FUNCTION_BLOCK FB_StrategyController_noChiller
VAR_INPUT
	ambientState : ST_AmbientState;
	
	//actual temperatures in thermal networks
	cnState : ST_ThermalNetworkState;
	hnltState : ST_ThermalNetworkState;
	hnhtState : ST_ThermalNetworkState;
END_VAR
VAR_OUTPUT	
	cnControl : ST_CoolingNetworkControl;
	hnltControl : ST_HeatingNetworkLowTemperatureControl;	
	hnhtControl : ST_HeatingNetworkHighTemperatureControl;
	hnltCnLinkageControl : ST_HnltCnLinkageControl;
	hnhtHnltLinkageControl : ST_HnhtHnltLinkageControl;
	hnhtCnLinkageControl : ST_HnhtCnLinkageControl;
END_VAR
VAR
	{attribute 'OPC.UA.DA' := '1'}
	localSetParameters : ST_StrategySetParameters;	
	{attribute 'OPC.UA.DA' := '1'}
	localState : ST_StrategyState;	

	//default parameters
	localDefaultParameters : ST_StrategyDefaultParameters;

	//internal variables
	fTargetTemperature_HNHT_Heating : REAL;
	fTargetTemperature_HNHT_Cooling : REAL;
	fTargetTemperature_HNLT_Cooling : REAL;
	fTargetTemperature_HNLT_Heating : REAL;
	fTargetTemperature_CN : REAL;
	aTemperatureLimits_HNHT : ARRAY[1..2] OF REAL;
	aTemperatureLimits_HNLT : ARRAY[1..2] OF REAL;
	aTemperatureLimits_CN : ARRAY[1..2] OF REAL;
	stHNHTCheckDefaultParameters : ST_RangeCheckDefaultParameters := (tTaskCycleTime := GlobalVariables.tCtrlCycleTime_MAIN, tCtrlCycleTime := GlobalVariables.tCtrlCycleTime_MAIN, fRestoreDifference := 5);
	HNHT_Check : FB_RangeCheck := (ST_DefaultParameters := stHNHTCheckDefaultParameters);
	stHNLTCheckDefaultParameters : ST_RangeCheckDefaultParameters := (tTaskCycleTime := GlobalVariables.tCtrlCycleTime_MAIN, tCtrlCycleTime := GlobalVariables.tCtrlCycleTime_MAIN, fRestoreDifference := 5);
	HNLT_Check : FB_RangeCheck := (ST_DefaultParameters := stHNLTCheckDefaultParameters);
	stCNCheckDefaultParameters : ST_RangeCheckDefaultParameters := (tTaskCycleTime := GlobalVariables.tCtrlCycleTime_MAIN, tCtrlCycleTime := GlobalVariables.tCtrlCycleTime_MAIN, fRestoreDifference := 2);
	CN_Check : FB_RangeCheck := (ST_DefaultParameters := stCNCheckDefaultParameters);
	
	
	//controller and variables for high temperature heating network
	fOffset_TargetTemperature_CHP1 : REAL; //not fixed, switches depending on ambient temperature -> see method: ControlHNHT
	fOffset_TargetTemperature_CHP2 : REAL; //not fixed, switches depending on ambient temperature -> see method: ControlHNHT
	Controller_CHP_Prioritization : FB_CTRL_2POINT;
	Controller_CHP_Prioritization_Parameters : ST_CTRL_2POINT_PARAMS;	
	Controller_CHP1_UpperTemperature : FB_CTRL_2POINT; //check upper temperature for turning on chp
	Controller_CHP1_LowerTemperature : FB_CTRL_2POINT; //check lower temperature for turning off chp
	Controller_CHP1_Parameters : ST_CTRL_2POINT_PARAMS;	
	Trigger_CHP1_UpperTemperature : F_TRIG;
	Trigger_CHP1_LowerTemperature : F_TRIG;
	bTrigger_CHP1 : BOOL;
	Controller_CHP2_UpperTemperature : FB_CTRL_2POINT;
	Controller_CHP2_LowerTemperature : FB_CTRL_2POINT;
	Controller_CHP2_Parameters : ST_CTRL_2POINT_PARAMS;
	Trigger_CHP2_UpperTemperature : F_TRIG;
	Trigger_CHP2_LowerTemperature : F_TRIG;
	bTrigger_CHP2 : BOOL;
	Controller_CondensingBoiler : FB_CTRL_2POINT;
	Controller_CondensingBoiler_Parameters : ST_CTRL_2POINT_PARAMS;
	Controller_VSI_Loading_Permission : FB_CTRL_2POINT;
	Controller_VSI_Loading_Permission_Parameters : ST_CTRL_2POINT_PARAMS;
	Controller_VSI_Unloading_Permission : FB_CTRL_2POINT;
	Controller_VSI_Unloading_Permission_Parameters : ST_CTRL_2POINT_PARAMS;
	Controller_Buffer_VSI_Unloading : FB_CTRL_2POINT;
	Controller_Buffer_VSI_Unloading_Parameters : ST_CTRL_2POINT_PARAMS;
	Controller_StaticHeating : FB_CTRL_2POINT;
	Controller_StaticHeating_Parameters : ST_CTRL_2POINT_PARAMS;
	
	//controllers and variables for low temperature heating network
	Controller_OuterCapillaryTubeMats : FB_CTRL_2POINT;
	Controller_OuterCapillaryTubeMats_Parameters : ST_CTRL_2POINT_PARAMS;
	Controller_OuterCapillaryTubeMats_Permission : FB_CTRL_2POINT;
	Controller_OuterCapillaryTubeMats_Permission_Parameters : ST_CTRL_2POINT_PARAMS;
	fOffset_TargetTemperature_OuterCapillaryTubeMats_Cooling : REAL := 1;	
	fOffset_OuterCapillaryTubeMats_Permission : REAL := 10;
	
	Controller_HVFA_HNLT_HVFALoadingPermission : FB_CTRL_2POINT;
	Controller_HVFA_HNLT_HVFALoadingPermission_Parameters : ST_CTRL_2POINT_PARAMS;
	Controller_HVFA_HNLT_HVFAUnloadingPermission : FB_CTRL_2POINT;
	Controller_HVFA_HNLT_HVFAUnloadingPermission_Parameters : ST_CTRL_2POINT_PARAMS;
	Controller_Buffer_HVFA_HNLT_HVFAUnloading : FB_CTRL_2POINT;
	Controller_Buffer_HVFA_HNLT_HVFAUnloading_Parameters : ST_CTRL_2POINT_PARAMS;
	Controller_Buffer_HVFA_HNLT_HVFALoading : FB_CTRL_2POINT;
	Controller_Buffer_HVFA_HNLT_HVFALoading_Parameters : ST_CTRL_2POINT_PARAMS;
	Controller_HVFA_HNLT_Recooling : FB_CTRL_2POINT;
	Controller_HVFA_HNLT_Recooling_Parameters : ST_CTRL_2POINT_PARAMS;
	fOffset_TargetTemperature_HVFA_HNLT_Heating : REAL := 1;
	fOffset_HVFA_HNLT_Recooling : REAL := 2;
		
	
	//controllers and variables for cooling network
	fOffset_TargetTemperature_eChiller : REAL := 0.5;	
	fOffset_TargetTemperature_HVFA_CN : REAL := 1;
	fOffset_TargetTemperature_HVFA_CN_Permission : REAL := 2.5;
	Controller_eChiller : FB_CTRL_2POINT;
	Controller_eChiller_Parameters : ST_CTRL_2POINT_PARAMS;	
	Controller_HVFA_CN_LoadingPermission : FB_CTRL_2POINT;
	Controller_HVFA_CN_LoadingPermission_Parameters : ST_CTRL_2POINT_PARAMS;
	Controller_HVFA_CN_UnloadingPermission : FB_CTRL_2POINT;
	Controller_HVFA_CN_UnloadingPermission_Parameters : ST_CTRL_2POINT_PARAMS;
	Controller_Buffer_HVFA_CN_Unloading : FB_CTRL_2POINT;
	Controller_Buffer_HVFA_CN_Unloading_Parameters : ST_CTRL_2POINT_PARAMS;

	//controllers and variables for hnht and hnlt linkage
	Controller_HeatExchanger1 : FB_CTRL_2POINT;
	Controller_HeatExchanger1_Parameters : ST_CTRL_2POINT_PARAMS;
	fOffset_TargetTemperature_HeatExchanger1 : REAL := 2;
	Controller_HeatPump_HNHT : FB_CTRL_2POINT;
	Controller_HeatPump_HNHT_Parameters : ST_CTRL_2POINT_PARAMS;
	fOffset_TargetTemperature_HeatPump_HNHT : REAL := 1;
	Controller_HeatPump_HNHT_Permission : FB_CTRL_2POINT;
	Controller_HeatPump_HNHT_Permission_Parameters : ST_CTRL_2POINT_PARAMS;
	fOffset_TargetTemperature_HeatPump_HNHT_Permission : REAL := 1;
	
	//controllers and variables for hnlt and cn linkage
	fOffset_TargetTemperature_HeatPump : REAL;
	Controller_HeatPump : FB_CTRL_2POINT;
	Controller_HeatPump_Parameters : ST_CTRL_2POINT_PARAMS;		

	//clock
	stDefaultParameters_Clock : ST_ClockDefaultParameters := (tTaskCycleTime := GlobalVariables.tCtrlCycleTime_MAIN, tCtrlCycleTime := T#1M);
	Clock : FB_Clock := (ST_DefaultParameters := stDefaultParameters_Clock);
END_VAR

Clock();
AmbientControl();
SetTemperatures();
ControlCN();
ControlHNLT();
ControlHNHT();
ControlHnltCnLinkage();
ControlHnhtHnltLinkage();
SetState();

METHOD AmbientControl : BOOL
VAR_INPUT
END_VAR
//check for heating or cooling mode
IF Clock.stClockState.sintMonth>4 AND Clock.stClockState.sintMonth<10 THEN
	//heating mode
	hnltCnLinkageControl.bHeatingMode := FALSE;
	hnhtCnLinkageControl.bHeatingMode := FALSE;
ELSE
	//cooling mode	
	hnltCnLinkageControl.bHeatingMode := TRUE;
	hnhtCnLinkageControl.bHeatingMode := TRUE;
END_IF
END_METHOD

METHOD ControlCN : BOOL
VAR_INPUT
END_VAR
//set hysteresis parameters for two-point controllers in cooling network
Controller_eChiller_Parameters.fHysteresisRange := 7;
Controller_eChiller_Parameters.tCtrlCycleTime := GlobalVariables.tCtrlCycleTime_MAIN;
Controller_eChiller_Parameters.tTaskCycleTime := GlobalVariables.tTaskCycleTime_MAIN;

//permission to load storage depending on upper hvfa storage temperature
Controller_HVFA_CN_LoadingPermission_Parameters.fHysteresisRange := 1;
Controller_HVFA_CN_LoadingPermission_Parameters.tCtrlCycleTime := GlobalVariables.tCtrlCycleTime_MAIN;
Controller_HVFA_CN_LoadingPermission_Parameters.tTaskCycleTime := GlobalVariables.tTaskCycleTime_MAIN;

//permission to unload storage depending on upper hvfa storage temperature
Controller_HVFA_CN_UnloadingPermission_Parameters.fHysteresisRange := 1;
Controller_HVFA_CN_UnloadingPermission_Parameters.tCtrlCycleTime := GlobalVariables.tCtrlCycleTime_MAIN;
Controller_HVFA_CN_UnloadingPermission_Parameters.tTaskCycleTime := GlobalVariables.tTaskCycleTime_MAIN;

//hysteresis for unloading hvfa storage depending on buffer storage temperature
Controller_Buffer_HVFA_CN_Unloading_Parameters.fHysteresisRange := 2;
Controller_Buffer_HVFA_CN_Unloading_Parameters.tCtrlCycleTime := GlobalVariables.tCtrlCycleTime_MAIN;
Controller_Buffer_HVFA_CN_Unloading_Parameters.tTaskCycleTime := GlobalVariables.tTaskCycleTime_MAIN;

//control eChiller
Controller_eChiller(fSetpointValue := cnState.fMidTemperature,
	fActualValue := fTargetTemperature_CN-fOffset_TargetTemperature_eChiller,
	eMode := eCTRL_MODE_ACTIVE,
	stParams := Controller_eChiller_Parameters);

//control hvfa storage loading permission 
Controller_HVFA_CN_LoadingPermission(fSetpointValue := cnState.fUpperTemperature_ActiveStorage,
	fActualValue := fTargetTemperature_CN-fOffset_TargetTemperature_HVFA_CN_Permission,
	eMode := eCTRL_MODE_ACTIVE,
	stParams := Controller_HVFA_CN_LoadingPermission_Parameters);
	
//control hvfa storage unloading permission 
Controller_HVFA_CN_UnloadingPermission(fSetpointValue := fTargetTemperature_CN-fOffset_TargetTemperature_HVFA_CN_Permission,
	fActualValue := cnState.fLowerTemperature_ActiveStorage,
	eMode := eCTRL_MODE_ACTIVE,
	stParams := Controller_HVFA_CN_UnloadingPermission_Parameters);
	
//unloading permission buffer HVFA
Controller_Buffer_HVFA_CN_Unloading(fSetpointValue := cnState.fMidTemperature,
	fActualValue := fTargetTemperature_CN+fOffset_TargetTemperature_HVFA_CN,
	eMode := eCTRL_MODE_ACTIVE,
	stParams := Controller_Buffer_HVFA_CN_Unloading_Parameters);
	
IF Clock.stClockState.sintMonth>4 AND Clock.stClockState.sintMonth<10 THEN
	cnControl.bSetStatusOn_eChiller := TRUE;
	cnControl.bSetStatusOn_HVFASystem := FALSE;
	cnControl.bLoading_HVFASystem := FALSE;
ELSE
	cnControl.bSetStatusOn_eChiller := Controller_eChiller.bOut;
	cnControl.bSetStatusOn_HVFASystem := (Controller_Buffer_HVFA_CN_Unloading.bOut AND Controller_HVFA_CN_UnloadingPermission.bOut) OR ((cnControl.bSetStatusOn_eChiller) AND NOT Controller_Buffer_HVFA_CN_Unloading.bOut AND Controller_HVFA_CN_LoadingPermission.bOut); 
	cnControl.bLoading_HVFASystem := NOT (Controller_Buffer_HVFA_CN_Unloading.bOut AND Controller_HVFA_CN_UnloadingPermission.bOut);
END_IF

cnControl.bSetStatusOn_eChiller := FALSE; //strategy without eChiller
cnControl.bSetStatusOn_HVFASystem := FALSE;
cnControl.bLoading_HVFASystem := FALSE;


//cnControl.bSetStatusOn_HVFASystem := FALSE;
//cnControl.bLoading_HVFASystem := FALSE;
END_METHOD

METHOD ControlHNHT : BOOL
VAR_INPUT
END_VAR
VAR
END_VAR
//set hysteresis parameters for two-point controllers in high temperature heating network
Controller_CHP_Prioritization_Parameters.fHysteresisRange := 4;
Controller_CHP_Prioritization_Parameters.tCtrlCycleTime := GlobalVariables.tCtrlCycleTime_MAIN;
Controller_CHP_Prioritization_Parameters.tTaskCycleTime := GlobalVariables.tTaskCycleTime_MAIN;

Controller_CHP1_Parameters.tCtrlCycleTime := GlobalVariables.tCtrlCycleTime_MAIN;
Controller_CHP1_Parameters.tTaskCycleTime := GlobalVariables.tTaskCycleTime_MAIN;
Controller_CHP2_Parameters.tCtrlCycleTime := GlobalVariables.tCtrlCycleTime_MAIN;
Controller_CHP2_Parameters.tTaskCycleTime := GlobalVariables.tTaskCycleTime_MAIN;

Controller_CondensingBoiler_Parameters.fHysteresisRange := 12;
Controller_CondensingBoiler_Parameters.tCtrlCycleTime := GlobalVariables.tCtrlCycleTime_MAIN;
Controller_CondensingBoiler_Parameters.tTaskCycleTime := GlobalVariables.tTaskCycleTime_MAIN;

Controller_Buffer_VSI_Unloading_Parameters.fHysteresisRange := 4;
Controller_Buffer_VSI_Unloading_Parameters.tCtrlCycleTime := GlobalVariables.tCtrlCycleTime_MAIN;
Controller_Buffer_VSI_Unloading_Parameters.tTaskCycleTime := GlobalVariables.tTaskCycleTime_MAIN;

Controller_VSI_Unloading_Permission_Parameters.fHysteresisRange := 4;
Controller_VSI_Unloading_Permission_Parameters.tCtrlCycleTime := GlobalVariables.tCtrlCycleTime_MAIN;
Controller_VSI_Unloading_Permission_Parameters.tTaskCycleTime := GlobalVariables.tTaskCycleTime_MAIN;

Controller_VSI_Loading_Permission_Parameters.fHysteresisRange := 4;
Controller_VSI_Loading_Permission_Parameters.tCtrlCycleTime := GlobalVariables.tCtrlCycleTime_MAIN;
Controller_VSI_Loading_Permission_Parameters.tTaskCycleTime := GlobalVariables.tTaskCycleTime_MAIN;

Controller_StaticHeating_Parameters.fHysteresisRange := 4;
Controller_StaticHeating_Parameters.tCtrlCycleTime := GlobalVariables.tCtrlCycleTime_MAIN;
Controller_StaticHeating_Parameters.tTaskCycleTime := GlobalVariables.tTaskCycleTime_MAIN;

Controller_CHP_Prioritization(fSetpointValue := 15,
	fActualValue := ambientState.fOutsideTemperature_Mean,
	eMode := eCTRL_MODE_ACTIVE,
	stParams := Controller_CHP_Prioritization_Parameters);
IF Controller_CHP_Prioritization.bOut THEN
	//prioritize large CHP (CHP2) during cold temperatures
	Controller_CHP1_Parameters.fHysteresisRange := 14;
	Controller_CHP2_Parameters.fHysteresisRange := 12;
	fOffset_TargetTemperature_CHP1 := 1;
	fOffset_TargetTemperature_CHP2 := 0;
ELSE
	//prioritize large CHP (CHP2) during cold temperatures
	Controller_CHP1_Parameters.fHysteresisRange := 12;
	Controller_CHP2_Parameters.fHysteresisRange := 14;	
	fOffset_TargetTemperature_CHP1 := 0;
	fOffset_TargetTemperature_CHP2 := 1;	
END_IF

//start when upper temperature too cold and stop when lower temperature too hot
Controller_CHP1_UpperTemperature(fSetpointValue := fTargetTemperature_HNHT_Heating-fOffset_TargetTemperature_CHP1,
	fActualValue := hnhtState.fUpperTemperature,
	eMode := eCTRL_MODE_ACTIVE,
	stParams := Controller_CHP1_Parameters);
Controller_CHP1_LowerTemperature(fSetpointValue := fTargetTemperature_HNHT_Heating-fOffset_TargetTemperature_CHP1,
	fActualValue := hnhtState.fLowerTemperature,
	eMode := eCTRL_MODE_ACTIVE,
	stParams := Controller_CHP1_Parameters);
Trigger_CHP1_UpperTemperature(CLK := Controller_CHP1_UpperTemperature.bOut);
Trigger_CHP1_LowerTemperature(CLK := Controller_CHP1_LowerTemperature.bOut);
IF Trigger_CHP1_UpperTemperature.Q THEN
	bTrigger_CHP1 := TRUE;
END_IF
IF Trigger_CHP1_LowerTemperature.Q THEN
	bTrigger_CHP1 := FALSE;
END_IF
hnhtControl.bSetStatusOn_CHP1 := Controller_CHP1_UpperTemperature.bOut OR (Controller_CHP1_LowerTemperature.bOut AND bTrigger_CHP1);

//start when upper temperature too cold and stop when lower temperature too hot
Controller_CHP2_UpperTemperature(fSetpointValue := fTargetTemperature_HNHT_Heating-fOffset_TargetTemperature_CHP2,
	fActualValue := hnhtState.fUpperTemperature,
	eMode := eCTRL_MODE_ACTIVE,
	stParams := Controller_CHP2_Parameters);
Controller_CHP2_LowerTemperature(fSetpointValue := fTargetTemperature_HNHT_Heating-fOffset_TargetTemperature_CHP2,
	fActualValue := hnhtState.fLowerTemperature,
	eMode := eCTRL_MODE_ACTIVE,
	stParams := Controller_CHP2_Parameters);
Trigger_CHP2_UpperTemperature(CLK := Controller_CHP2_UpperTemperature.bOut);
Trigger_CHP2_LowerTemperature(CLK := Controller_CHP2_LowerTemperature.bOut);
IF Trigger_CHP2_UpperTemperature.Q THEN
	bTrigger_CHP2 := TRUE;
END_IF
IF Trigger_CHP2_LowerTemperature.Q THEN
	bTrigger_CHP2 := FALSE;
END_IF
hnhtControl.bSetStatusOn_CHP2 := Controller_CHP2_UpperTemperature.bOut OR (Controller_CHP2_LowerTemperature.bOut AND bTrigger_CHP2);

Controller_CondensingBoiler(fSetpointValue := fTargetTemperature_HNHT_Heating,
	fActualValue := hnhtState.fUpperTemperature,
	eMode := eCTRL_MODE_ACTIVE,
	stParams := Controller_CondensingBoiler_Parameters);
hnhtControl.bSetStatusOn_CondensingBoiler := Controller_CondensingBoiler.bOut;

//buffer storage asks VSI for unloading when buffer storage temperature falls below limit
Controller_Buffer_VSI_Unloading(fSetpointValue := fTargetTemperature_HNHT_Heating,
	fActualValue := hnhtState.fUpperTemperature,
	eMode := eCTRL_MODE_ACTIVE,
	stParams := Controller_Buffer_VSI_Unloading_Parameters);

//VSI storage may only be unloaded when upper temperature is between limits for unloading
Controller_VSI_Unloading_Permission(fSetpointValue := hnhtState.fUpperTemperature_ActiveStorage,
	fActualValue := fTargetTemperature_HNHT_Heating,
	eMode := eCTRL_MODE_ACTIVE,
	stParams := Controller_VSI_Unloading_Permission_Parameters);
	
//VSI storage may only be loaded when lower temperature is between limits for loading
Controller_VSI_Loading_Permission(fSetpointValue := fTargetTemperature_HNHT_Heating,
	fActualValue := hnhtState.fLowerTemperature_ActiveStorage,
	eMode := eCTRL_MODE_ACTIVE,
	stParams := Controller_VSI_Loading_Permission_Parameters);
	
hnhtControl.bSetStatusOn_VSIStorage := (Controller_Buffer_VSI_Unloading.bOut AND Controller_VSI_Unloading_Permission.bOut) OR ((hnhtControl.bSetStatusOn_CHP1 OR hnhtControl.bSetStatusOn_CHP2) AND NOT Controller_Buffer_VSI_Unloading.bOut AND Controller_VSI_Loading_Permission.bOut); 
hnhtControl.bLoading_VSISystem := NOT (Controller_Buffer_VSI_Unloading.bOut AND Controller_VSI_Unloading_Permission.bOut);

//condensing boiler is switched if network temperature falls below critical temperature limit
Controller_StaticHeating(fSetpointValue := 15,
	fActualValue := ambientState.fOutsideTemperature,
	eMode := eCTRL_MODE_ACTIVE,
	stParams := Controller_StaticHeating_Parameters);
hnhtControl.bSetStatusOn_StaticHeating := Controller_StaticHeating.bOut;
END_METHOD

METHOD ControlHnhtHnltLinkage : BOOL
VAR_INPUT
END_VAR
Controller_HeatExchanger1_Parameters.fHysteresisRange := 8;
Controller_HeatExchanger1_Parameters.tCtrlCycleTime := GlobalVariables.tCtrlCycleTime_MAIN;
Controller_HeatExchanger1_Parameters.tTaskCycleTime := GlobalVariables.tTaskCycleTime_MAIN;

Controller_HeatPump_HNHT_Parameters.fHysteresisRange := 10;
Controller_HeatPump_HNHT_Parameters.tCtrlCycleTime := GlobalVariables.tCtrlCycleTime_MAIN;
Controller_HeatPump_HNHT_Parameters.tTaskCycleTime := GlobalVariables.tTaskCycleTime_MAIN;

Controller_HeatPump_HNHT_Permission_Parameters.fHysteresisRange := 4;
Controller_HeatPump_HNHT_Permission_Parameters.tCtrlCycleTime := GlobalVariables.tCtrlCycleTime_MAIN;
Controller_HeatPump_HNHT_Permission_Parameters.tTaskCycleTime := GlobalVariables.tTaskCycleTime_MAIN;

//control heat exchanger 1
Controller_HeatExchanger1(fSetpointValue := fTargetTemperature_HNLT_Heating-fOffset_TargetTemperature_HeatExchanger1,
	fActualValue := hnltState.fMidTemperature,
	eMode := eCTRL_MODE_ACTIVE,
	stParams := Controller_HeatExchanger1_Parameters);
hnhtHnltLinkageControl.bSetStatusOn_HeatExchanger1 := Controller_HeatExchanger1.bOut;

//control heat pump hnht
Controller_HeatPump_HNHT(fSetpointValue := fTargetTemperature_HNHT_Heating+fOffset_TargetTemperature_HeatPump_HNHT,
	fActualValue := hnhtState.fUpperTemperature,
	eMode := eCTRL_MODE_ACTIVE,
	stParams := Controller_HeatPump_HNHT_Parameters);
	
Controller_HeatPump_HNHT_Permission(fSetpointValue := hnltState.fMidTemperature,
	fActualValue := fTargetTemperature_HNLT_Cooling+fOffset_TargetTemperature_HeatPump_HNHT_Permission,
	eMode := eCTRL_MODE_ACTIVE,
	stParams := Controller_HeatPump_HNHT_Permission_Parameters);	
	
// HP currently only able to reach 65°C flow temperature (hard-coded HP-internal)
// IF localSetParameters.bProductionModeActivated THEN
// 	hnhtHnltLinkageControl.bSetStatusOn_HeatPump := FALSE;
// ELSE
// 	hnhtHnltLinkageControl.bSetStatusOn_HeatPump := Controller_HeatPump_HNHT.bOut AND Controller_HeatPump_HNHT_Permission.bOut;
// END_IF

// When using a heating target temp of 60 °C in production mode the heat pump can be used in both operating modes
hnhtHnltLinkageControl.bSetStatusOn_HeatPump := Controller_HeatPump_HNHT.bOut AND Controller_HeatPump_HNHT_Permission.bOut;
END_METHOD

METHOD ControlHNLT : BOOL
VAR_INPUT
END_VAR
//set hysteresis parameters for two-point controllers in cooling network
Controller_OuterCapillaryTubeMats_Parameters.fHysteresisRange := 6;
Controller_OuterCapillaryTubeMats_Parameters.tCtrlCycleTime := GlobalVariables.tCtrlCycleTime_MAIN;
Controller_OuterCapillaryTubeMats_Parameters.tTaskCycleTime := GlobalVariables.tTaskCycleTime_MAIN;

Controller_OuterCapillaryTubeMats_Permission_Parameters.fHysteresisRange := 6;
Controller_OuterCapillaryTubeMats_Permission_Parameters.tCtrlCycleTime := GlobalVariables.tCtrlCycleTime_MAIN;
Controller_OuterCapillaryTubeMats_Permission_Parameters.tTaskCycleTime := GlobalVariables.tTaskCycleTime_MAIN;


//control strategy for cooling network - fSetpointValue and fActualValue are changed for cooling applications
Controller_OuterCapillaryTubeMats(fSetpointValue := hnltState.fMidTemperature,
	fActualValue := fTargetTemperature_HNLT_Cooling+fOffset_TargetTemperature_OuterCapillaryTubeMats_Cooling,
	eMode := eCTRL_MODE_ACTIVE,
	stParams := Controller_OuterCapillaryTubeMats_Parameters);

//permission controller to ensure that network ist not heated up if ambient temperature is too high
Controller_OuterCapillaryTubeMats_Permission(fSetpointValue := fTargetTemperature_HNLT_Cooling-fOffset_OuterCapillaryTubeMats_Permission,
	fActualValue := ambientState.fOutsideTemperature,
	eMode := eCTRL_MODE_ACTIVE,
	stParams := Controller_OuterCapillaryTubeMats_Permission_Parameters);

//control hvfa storage
//set hysteresis parameters for two-point controllers in low temperature heating network

Controller_Buffer_HVFA_HNLT_HVFAUnloading_Parameters.fHysteresisRange := 6;
Controller_Buffer_HVFA_HNLT_HVFAUnloading_Parameters.tCtrlCycleTime := GlobalVariables.tCtrlCycleTime_MAIN;
Controller_Buffer_HVFA_HNLT_HVFAUnloading_Parameters.tTaskCycleTime := GlobalVariables.tTaskCycleTime_MAIN;

Controller_Buffer_HVFA_HNLT_HVFALoading_Parameters.fHysteresisRange := 4;
Controller_Buffer_HVFA_HNLT_HVFALoading_Parameters.tCtrlCycleTime := GlobalVariables.tCtrlCycleTime_MAIN;
Controller_Buffer_HVFA_HNLT_HVFALoading_Parameters.tTaskCycleTime := GlobalVariables.tTaskCycleTime_MAIN;

Controller_HVFA_HNLT_Recooling_Parameters.fHysteresisRange := 4;
Controller_HVFA_HNLT_Recooling_Parameters.tCtrlCycleTime := GlobalVariables.tCtrlCycleTime_MAIN;
Controller_HVFA_HNLT_Recooling_Parameters.tTaskCycleTime := GlobalVariables.tTaskCycleTime_MAIN;

Controller_HVFA_HNLT_HVFAUnloadingPermission_Parameters.fHysteresisRange := 4;
Controller_HVFA_HNLT_HVFAUnloadingPermission_Parameters.tCtrlCycleTime := GlobalVariables.tCtrlCycleTime_MAIN;
Controller_HVFA_HNLT_HVFAUnloadingPermission_Parameters.tTaskCycleTime := GlobalVariables.tTaskCycleTime_MAIN;

Controller_HVFA_HNLT_HVFALoadingPermission_Parameters.fHysteresisRange := 4;
Controller_HVFA_HNLT_HVFALoadingPermission_Parameters.tCtrlCycleTime := GlobalVariables.tCtrlCycleTime_MAIN;
Controller_HVFA_HNLT_HVFALoadingPermission_Parameters.tTaskCycleTime := GlobalVariables.tTaskCycleTime_MAIN;

//buffer storage asks HVFA_HNLT for unloading when buffer storage temperature falls below limit
Controller_Buffer_HVFA_HNLT_HVFAUnloading(fSetpointValue := fTargetTemperature_HNLT_Heating-fOffset_TargetTemperature_HVFA_HNLT_Heating,
	fActualValue := hnltState.fMidTemperature,
	eMode := eCTRL_MODE_ACTIVE,
	stParams := Controller_Buffer_HVFA_HNLT_HVFAUnloading_Parameters);
	
//buffer storage asks HVFA_HNLT for loading when buffer storage temperature rises above limit
Controller_Buffer_HVFA_HNLT_HVFALoading(fSetpointValue := hnltState.fMidTemperature,
	fActualValue := fTargetTemperature_HNLT_Cooling,
	eMode := eCTRL_MODE_ACTIVE,
	stParams := Controller_Buffer_HVFA_HNLT_HVFALoading_Parameters);

//hvfa storage may only be unloaded when upper temperature is between limits for unloading
Controller_HVFA_HNLT_HVFAUnloadingPermission(fSetpointValue := hnltState.fLowerTemperature_ActiveStorage,
	fActualValue := fTargetTemperature_HNLT_Heating,
	eMode := eCTRL_MODE_ACTIVE,
	stParams := Controller_HVFA_HNLT_HVFAUnloadingPermission_Parameters);
	
//hvfa storage may only be loaded when lower temperature is between limits for loading
Controller_HVFA_HNLT_HVFALoadingPermission(fSetpointValue := fTargetTemperature_HNLT_Cooling,
	fActualValue := hnltState.fLowerTemperature_ActiveStorage,
	eMode := eCTRL_MODE_ACTIVE,
	stParams := Controller_HVFA_HNLT_HVFALoadingPermission_Parameters);

//enable hvfa recooling during low temperature times in summer months	
Controller_HVFA_HNLT_Recooling(fSetpointValue := hnltState.fLowerTemperature_ActiveStorage,
	fActualValue := fTargetTemperature_HNLT_Cooling-fOffset_HVFA_HNLT_Recooling,
	eMode := eCTRL_MODE_ACTIVE,
	stParams := Controller_HVFA_HNLT_Recooling_Parameters);
	
IF hnltCnLinkageControl.bHeatingMode THEN
	hnltControl.bSetStatusOn_HVFASystem := (Controller_HVFA_HNLT_HVFALoadingPermission.bOut AND Controller_Buffer_HVFA_HNLT_HVFALoading.bOut) OR (Controller_HVFA_HNLT_HVFAUnloadingPermission.bOut AND Controller_Buffer_HVFA_HNLT_HVFAUnloading.bOut);
	hnltControl.bLoading_HVFASystem := Controller_HVFA_HNLT_HVFALoadingPermission.bOut AND Controller_Buffer_HVFA_HNLT_HVFALoading.bOut;
	hnltControl.bSetStatusOn_OuterCapillaryTubeMats := Controller_OuterCapillaryTubeMats.bOut AND Controller_OuterCapillaryTubeMats_Permission.bOut;
ELSE
	hnltControl.bSetStatusOn_HVFASystem := ((Controller_HVFA_HNLT_HVFALoadingPermission.bOut AND Controller_Buffer_HVFA_HNLT_HVFALoading.bOut) OR (Controller_HVFA_HNLT_HVFAUnloadingPermission.bOut AND Controller_Buffer_HVFA_HNLT_HVFAUnloading.bOut)) OR (Controller_HVFA_HNLT_Recooling.bOut AND Controller_OuterCapillaryTubeMats_Permission.bOut);
	hnltControl.bLoading_HVFASystem := Controller_HVFA_HNLT_HVFALoadingPermission.bOut AND Controller_Buffer_HVFA_HNLT_HVFALoading.bOut;
	hnltControl.bSetStatusOn_OuterCapillaryTubeMats := (Controller_OuterCapillaryTubeMats.bOut AND Controller_OuterCapillaryTubeMats_Permission.bOut) OR (Controller_HVFA_HNLT_Recooling.bOut AND Controller_OuterCapillaryTubeMats_Permission.bOut);
END_IF
END_METHOD

METHOD ControlHnltCnLinkage : BOOL
VAR_INPUT
END_VAR
//set hysteresis parameters for hnlt cn linkage systems
fOffset_TargetTemperature_HeatPump := 0;
Controller_HeatPump_Parameters.fHysteresisRange := 4;
Controller_HeatPump_Parameters.tCtrlCycleTime := GlobalVariables.tCtrlCycleTime_MAIN;
Controller_HeatPump_Parameters.tTaskCycleTime := GlobalVariables.tTaskCycleTime_MAIN;
	
//control heat pump depending on heating demand in hnlt

Controller_HeatPump(fSetpointValue := cnState.fMidTemperature,
	fActualValue := fTargetTemperature_CN,
	eMode := eCTRL_MODE_ACTIVE,
	stParams := Controller_HeatPump_Parameters);
	
hnltCnLinkageControl.bSetStatusOn_HeatPump := Controller_HeatPump.bOut;

hnltCnLinkageControl.fTargetTemperature_ProductionHall := localDefaultParameters.fTargetTemperature_ProductionHall;

hnltCnLinkageControl.bSetStatusOn_InnerCapillaryTubeMats := FALSE; //turn off cooling when eChiller is not available
hnltCnLinkageControl.bSetStatusOn_UnderfloorHeating := FALSE; //turn off cooling when eChiller is not available
END_METHOD

METHOD SetState : BOOL
VAR_INPUT
END_VAR
localState.fTargetTemperature_HNHT_Heating := fTargetTemperature_HNHT_Heating;
localState.fTargetTemperature_HNHT_Cooling := fTargetTemperature_HNHT_Cooling;
localState.fTargetTemperature_HNLT_Heating := fTargetTemperature_HNLT_Heating;
localState.fTargetTemperature_HNLT_Cooling := fTargetTemperature_HNLT_Cooling;
localState.fTargetTemperature_CN := fTargetTemperature_CN;
localState.fTargetTemperature_ProductionHall := localDefaultParameters.fTargetTemperature_ProductionHall;

localState.aTemperatureLimits_HNHT := aTemperatureLimits_HNHT;
localState.aTemperatureLimits_HNLT := aTemperatureLimits_HNLT;
localState.aTemperatureLimits_CN := aTemperatureLimits_CN;	

localState.fFeedTemperature_HNHT := fTargetTemperature_HNHT_Heating+localDefaultParameters.fOffset_FeedTemperature_HNHT;
localState.fFeedTemperature_HNLT_Heating := fTargetTemperature_HNLT_Heating+localDefaultParameters.fOffset_FeedTemperature_HNLT_Heating;
localState.fFeedTemperature_HNLT_Cooling := fTargetTemperature_HNLT_Cooling-localDefaultParameters.fOffset_FeedTemperature_HNLT_Cooling;
localState.fFeedTemperature_CN := fTargetTemperature_CN-localDefaultParameters.fOffset_FeedTemperature_CN;
END_METHOD

METHOD SetTemperatures : BOOL
VAR_INPUT
END_VAR
//set internal variables depending on prodution mode
IF localSetParameters.bProductionModeActivated THEN
	IF Clock.stClockState.sintMonth>4 AND Clock.stClockState.sintMonth<10 THEN	
		fTargetTemperature_CN := localDefaultParameters.fTargetTemperature_CN_ProductionMode_Summer;
	ELSE
		fTargetTemperature_CN := localDefaultParameters.fTargetTemperature_CN_ProductionMode_Winter;
	END_IF
	fTargetTemperature_HNLT_Heating := localDefaultParameters.fTargetTemperature_HNLT_Heating_ProductionMode;
	fTargetTemperature_HNLT_Cooling := localDefaultParameters.fTargetTemperature_HNLT_Cooling_ProductionMode;
	fTargetTemperature_HNHT_Heating := localDefaultParameters.fTargetTemperature_HNHT_Heating_ProductionMode;
	fTargetTemperature_HNHT_Cooling := localDefaultParameters.fTargetTemperature_HNHT_Cooling_ProductionMode;
	aTemperatureLimits_CN := localDefaultParameters.aTemperatureLimits_CN_ProductionMode;
	aTemperatureLimits_HNLT := localDefaultParameters.aTemperatureLimits_HNLT_ProductionMode;
	aTemperatureLimits_HNHT := localDefaultParameters.aTemperatureLimits_HNHT_ProductionMode;

ELSE
	IF Clock.stClockState.sintMonth>4 AND Clock.stClockState.sintMonth<10 THEN	
		fTargetTemperature_CN := localDefaultParameters.fTargetTemperature_CN_Summer;
	ELSE
		fTargetTemperature_CN := localDefaultParameters.fTargetTemperature_CN_Winter;
	END_IF
	fTargetTemperature_HNLT_Heating := localDefaultParameters.fTargetTemperature_HNLT_Heating;
	fTargetTemperature_HNLT_Cooling := localDefaultParameters.fTargetTemperature_HNLT_Cooling;
	fTargetTemperature_HNHT_Heating := localDefaultParameters.fTargetTemperature_HNHT_Heating;
	fTargetTemperature_HNHT_Cooling := localDefaultParameters.fTargetTemperature_HNHT_Cooling;
	aTemperatureLimits_CN := localDefaultParameters.aTemperatureLimits_CN;
	aTemperatureLimits_HNLT := localDefaultParameters.aTemperatureLimits_HNLT;
	aTemperatureLimits_HNHT := localDefaultParameters.aTemperatureLimits_HNHT;
END_IF

//set feed temperatures
hnhtControl.fFeedTemperature := fTargetTemperature_HNHT_Heating+localDefaultParameters.fOffset_FeedTemperature_HNHT;
hnltControl.fFeedTemperature_Heating := fTargetTemperature_HNLT_Heating+localDefaultParameters.fOffset_FeedTemperature_HNLT_Heating;
hnltControl.fFeedTemperature_Cooling := fTargetTemperature_HNLT_Cooling-localDefaultParameters.fOffset_FeedTemperature_HNLT_Cooling;
cnControl.fFeedTemperature := fTargetTemperature_CN-localDefaultParameters.fOffset_FeedTemperature_CN;
hnhtHnltLinkageControl.fFeedTemperature_HNHT := hnhtControl.fFeedTemperature;
hnhtHnltLinkageControl.fFeedTemperature_HNLT_Heating := hnltControl.fFeedTemperature_Heating;
hnhtHnltLinkageControl.fFeedTemperature_HNLT_Cooling := hnltControl.fFeedTemperature_Cooling;
hnltCnLinkageControl.fFeedTemperature_CN := cnControl.fFeedTemperature;
hnltCnLinkageControl.fFeedTemperature_HNLT_Heating := hnltControl.fFeedTemperature_Heating;
hnltCnLinkageControl.fFeedTemperature_HNLT_Cooling := hnltControl.fFeedTemperature_Cooling;

//set algorithm permission depending on production mode to control structs
CN_Check(fInput := cnState.fMidTemperature,
	fLowerLimit := aTemperatureLimits_CN[1],
	fUpperLimit := aTemperatureLimits_CN[2]);
cnControl.bAlgorithmPermission := CN_Check.bPermission;
	
HNLT_Check(fInput := hnltState.fMidTemperature,
	fLowerLimit := aTemperatureLimits_HNLT[1],
	fUpperLimit := aTemperatureLimits_HNLT[2]);
hnltControl.bAlgorithmPermission := HNLT_Check.bPermission;
	
HNHT_Check(fInput := hnhtState.fMidTemperature,
	fLowerLimit := aTemperatureLimits_HNHT[1],
	fUpperLimit := aTemperatureLimits_HNHT[2]);	
hnhtControl.bAlgorithmPermission := HNHT_Check.bPermission;
	
hnltCnLinkageControl.bAlgorithmPermission_CN := cnControl.bAlgorithmPermission;
hnltCnLinkageControl.bAlgorithmPermission_HNLT := hnltControl.bAlgorithmPermission;
hnhtHnltLinkageControl.bAlgorithmPermission_HNHT := hnhtControl.bAlgorithmPermission;
hnhtHnltLinkageControl.bAlgorithmPermission_HNLT := hnltControl.bAlgorithmPermission;
hnhtCnLinkageControl.bAlgorithmPermission_CN := cnControl.bAlgorithmPermission;
hnhtCnLinkageControl.bAlgorithmPermission_HNHT := hnhtControl.bAlgorithmPermission;
END_METHOD

END_FUNCTION_BLOCK

(* stored: Version 1.1.0.1, ProductVersion 3.1.4024.10
   POU FB_StrategyController_noChiller: Id {5e2ad52c-f6b8-4c34-b0cd-c9904efa0df4}, SpecialFunc None
   Method AmbientControl: Id {8c83e0be-c123-4fd1-ab21-81ed7b9fab8e}
   Method ControlCN: Id {dec9fe09-afdc-4e4c-a1f2-0c0a5a108490}
   Method ControlHNHT: Id {a6883e4e-c7ec-4661-adae-d6c020e2e89b}
   Method ControlHnhtHnltLinkage: Id {01d836c6-ec43-4c40-bd4d-ef946a76be8f}
   Method ControlHNLT: Id {a237e22c-da97-4d13-9ce2-b4d3b0412fe8}
   Method ControlHnltCnLinkage: Id {350eeac8-30cf-40e9-8415-859c7473f1f5}
   Method SetState: Id {6ed24bee-b154-4f94-a576-52c05a559eb1}
   Method SetTemperatures: Id {1f1fa969-025a-4e33-bea9-d4c989259e20} *)
